// Mitsubishi GX Works2 project: MPS 장비 제어 7 (필수는 아님)   PLC: Q03UDV

PROGRAM MAIN
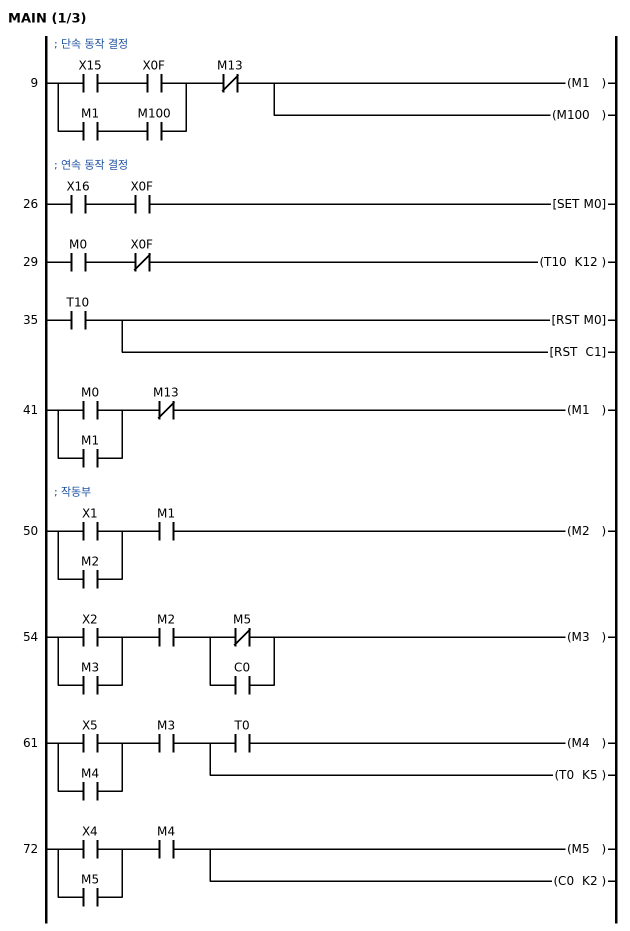
; 단속 동작 결정
9     LD      X15
      AND     X0F
      LD      M1
      AND     M100
      ORB
      ANI     M13
      OUT     M1
      OUT     M100
; 연속 동작 결정
26    LD      X16
      AND     X0F
      SET     M0
29    LD      M0
      ANI     X0F
      OUT     T10 K12
35    LD      T10
      RST     M0
      RST     C1
41    LD      M0
      OR      M1
      ANI     M13
      OUT     M1
; 작동부
50    LD      X1
      OR      M2
      AND     M1
      OUT     M2
54    LD      X2
      OR      M3
      AND     M2
      LDI     M5
      OR      C0
      ANB
      OUT     M3
61    LD      X5
      OR      M4
      AND     M3
      MPS
      AND     T0
      OUT     M4
      MPP
      OUT     T0 K5
72    LD      X4
      OR      M5
      AND     M4
      OUT     M5
      OUT     C0 K2
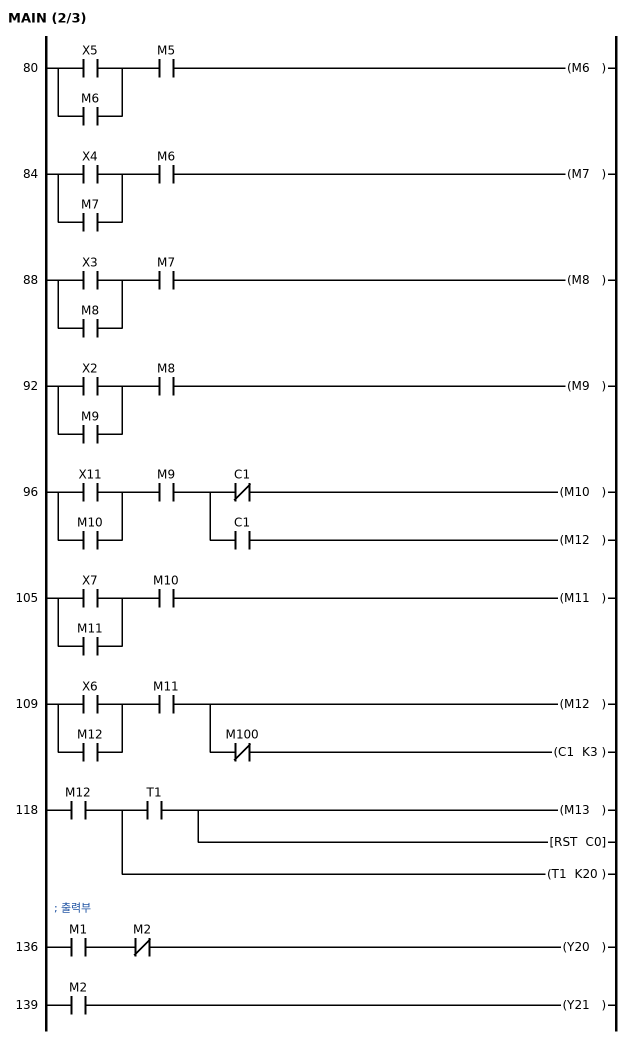
80    LD      X5
      OR      M6
      AND     M5
      OUT     M6
84    LD      X4
      OR      M7
      AND     M6
      OUT     M7
88    LD      X3
      OR      M8
      AND     M7
      OUT     M8
92    LD      X2
      OR      M9
      AND     M8
      OUT     M9
96    LD      X11
      OR      M10
      AND     M9
      MPS
      ANI     C1
      OUT     M10
      MPP
      AND     C1
      OUT     M12
105   LD      X7
      OR      M11
      AND     M10
      OUT     M11
109   LD      X6
      OR      M12
      AND     M11
      OUT     M12
      ANI     M100
      OUT     C1 K3
118   LD      M12
      MPS
      AND     T1
      OUT     M13
      RST     C0
      MPP
      OUT     T1 K20
; 출력부
136   LD      M1
      ANI     M2
      OUT     Y20
139   LD      M2
      OUT     Y21
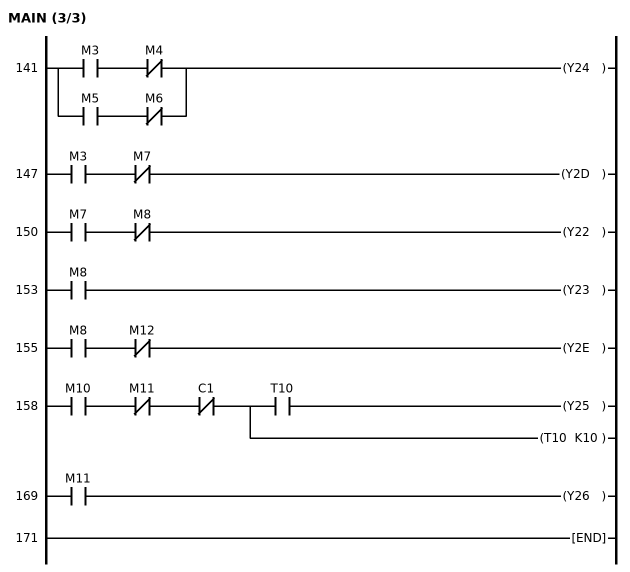
141   LD      M3
      ANI     M4
      LD      M5
      ANI     M6
      ORB
      OUT     Y24
147   LD      M3
      ANI     M7
      OUT     Y2D
150   LD      M7
      ANI     M8
      OUT     Y22
153   LD      M8
      OUT     Y23
155   LD      M8
      ANI     M12
      OUT     Y2E
158   LD      M10
      ANI     M11
      ANI     C1
      MPS
      AND     T10
      OUT     Y25
      MPP
      OUT     T10 K10
169   LD      M11
      OUT     Y26
171   END
END_PROGRAM
